FUNCTION_BLOCK TEST_TRIG (* Test trigonometric functions *)
  (* Standard: 61499-1 *)
  (* Version 0.0, 2006-09-05, JHC, Holobloc Inc *)
  (* Compiler header: package fb.rt.test; *)
  (* Compiler classdef: SimpleFB *)
  (* Compiler Java Sun JDK 1.5.0 *)
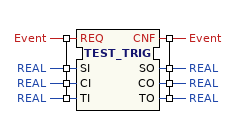
  EVENT_INPUT
    REQ WITH SI, CI, TI; (* Normal Execution Request *)
  END_EVENT
  EVENT_OUTPUT
    CNF WITH SO, CO, TO; (* Execution Confirmation *)
  END_EVENT
  VAR_INPUT
    SI : REAL; (* Input sin value *)
    CI : REAL; (* Input cos value *)
    TI : REAL; (* Input tan value *)
  END_VAR
  VAR_OUTPUT
    SO : REAL; (* sin(asin(SI)) *)
    CO : REAL; (* cos(acos(CI)) *)
    TO : REAL; (* tan(atan(TI)) *)
  END_VAR
  ALGORITHM REQ IN FBD: (* Normally executed algorithm *)
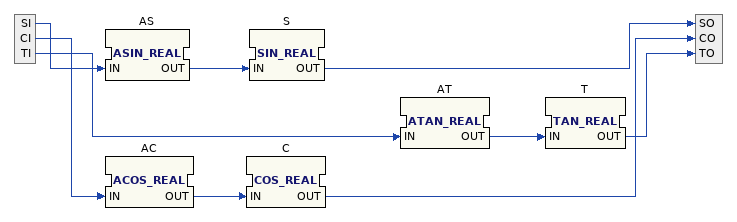
    FBS
      AS : ASIN_REAL;
      S : SIN_REAL;
      AC : ACOS_REAL;
      C : COS_REAL;
      AT : ATAN_REAL;
      T : TAN_REAL;
    END_FBS
    DATA_CONNECTIONS
      SI TO AS.IN;
      AS.OUT TO S.IN;
      S.OUT TO SO;
      CI TO AC.IN;
      AC.OUT TO C.IN;
      C.OUT TO CO;
      TI TO AT.IN;
      AT.OUT TO T.IN;
      T.OUT TO TO;
    END_CONNECTIONS
  END_ALGORITHM
END_FUNCTION_BLOCK
